// Mitsubishi GX Works2 project: js   PLC: Q02U
// js

PROGRAM MAIN
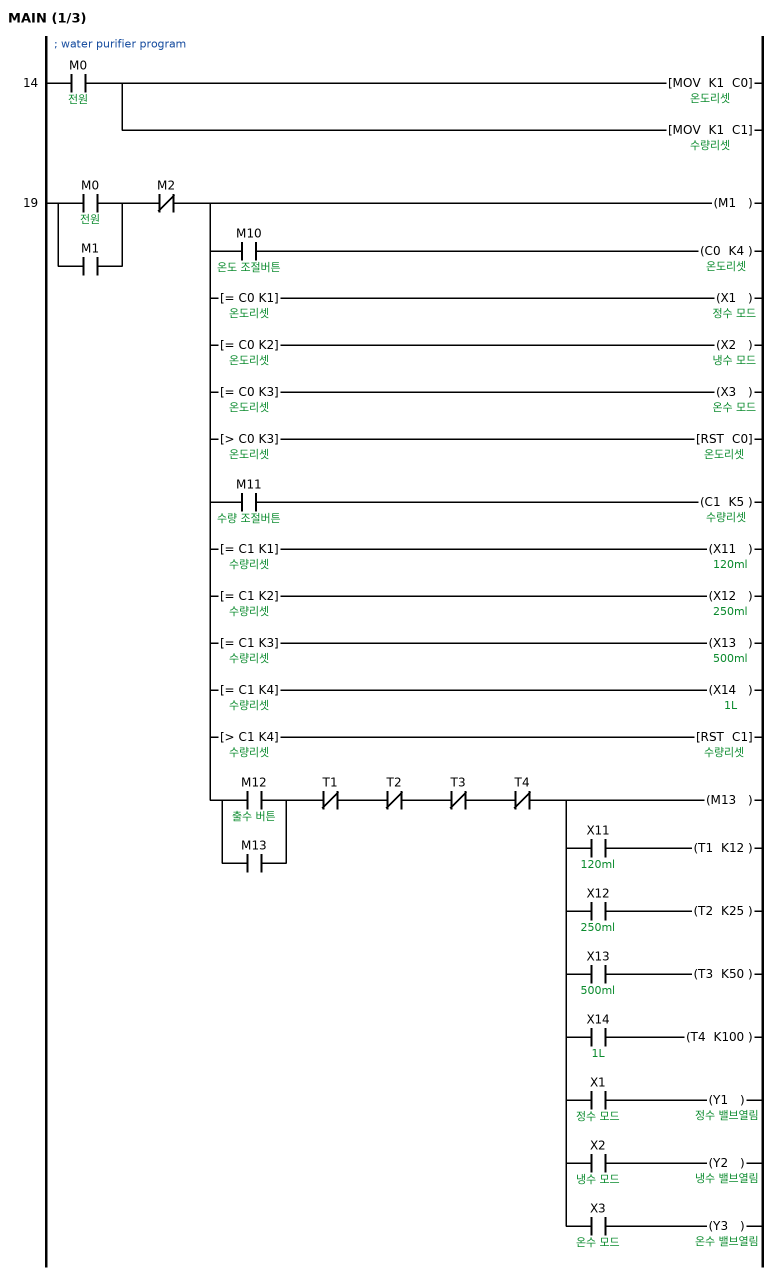
; water purifier program
14    LD      M0  ; 전원
      MOV     K1 C0  ; 온도리셋
      MOV     K1 C1  ; 수량리셋
19    LD      M0  ; 전원
      OR      M1
      ANI     M2
      OUT     M1
      MPS
      AND     M10  ; 온도 조절버튼
      OUT     C0 K4  ; 온도리셋
      MRD
      AND=    C0 K1  ; 온도리셋
      OUT     X1  ; 정수 모드
      MRD
      AND=    C0 K2  ; 온도리셋
      OUT     X2  ; 냉수 모드
      MRD
      AND=    C0 K3  ; 온도리셋
      OUT     X3  ; 온수 모드
      MRD
      AND>    C0 K3  ; 온도리셋
      RST     C0  ; 온도리셋
      MRD
      AND     M11  ; 수량 조절버튼
      OUT     C1 K5  ; 수량리셋
      MRD
      AND=    C1 K1  ; 수량리셋
      OUT     X11  ; 120ml
      MRD
      AND=    C1 K2  ; 수량리셋
      OUT     X12  ; 250ml
      MRD
      AND=    C1 K3  ; 수량리셋
      OUT     X13  ; 500ml
      MRD
      AND=    C1 K4  ; 수량리셋
      OUT     X14  ; 1L
      MRD
      AND>    C1 K4  ; 수량리셋
      RST     C1  ; 수량리셋
      MPP
      LD      M12  ; 출수 버튼
      OR      M13
      ANB
      ANI     T1
      ANI     T2
      ANI     T3
      ANI     T4
      OUT     M13
      MPS
      AND     X11  ; 120ml
      OUT     T1 K12
      MRD
      AND     X12  ; 250ml
      OUT     T2 K25
      MRD
      AND     X13  ; 500ml
      OUT     T3 K50
      MRD
      AND     X14  ; 1L
      OUT     T4 K100
      MRD
      AND     X1  ; 정수 모드
      OUT     Y1  ; 정수 밸브열림
      MRD
      AND     X2  ; 냉수 모드
      OUT     Y2  ; 냉수 밸브열림
      MPP
      AND     X3  ; 온수 모드
      OUT     Y3  ; 온수 밸브열림
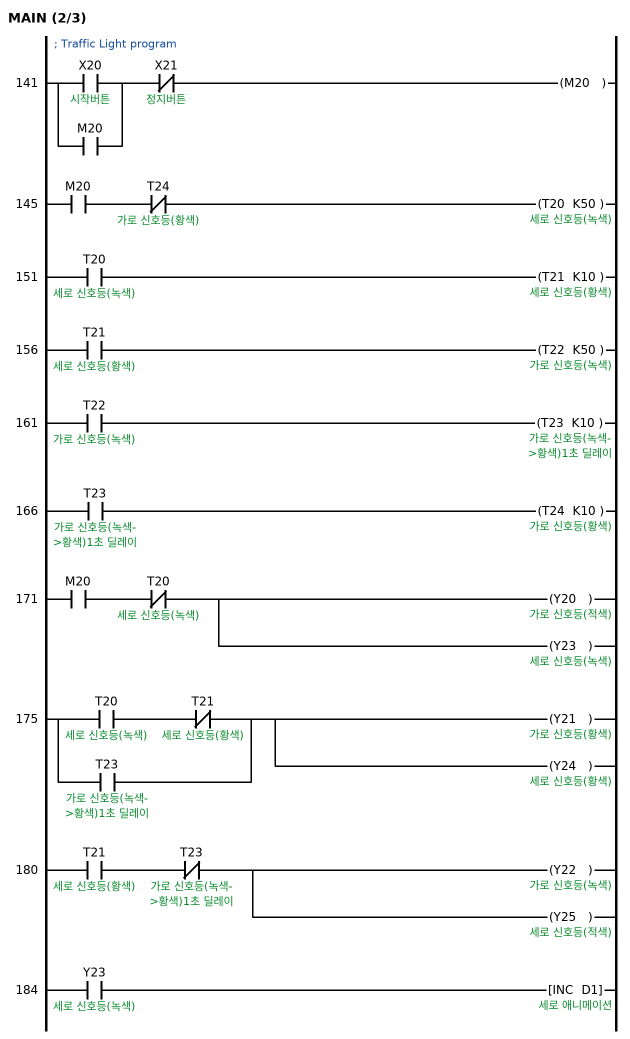
; Traffic Light program
141   LD      X20  ; 시작버튼
      OR      M20
      ANI     X21  ; 정지버튼
      OUT     M20
145   LD      M20
      ANI     T24  ; 가로 신호등(황색)
      OUT     T20 K50  ; 세로 신호등(녹색)
151   LD      T20  ; 세로 신호등(녹색)
      OUT     T21 K10  ; 세로 신호등(황색)
156   LD      T21  ; 세로 신호등(황색)
      OUT     T22 K50  ; 가로 신호등(녹색)
161   LD      T22  ; 가로 신호등(녹색)
      OUT     T23 K10  ; 가로 신호등(녹색->황색)1초 딜레이
166   LD      T23  ; 가로 신호등(녹색->황색)1초 딜레이
      OUT     T24 K10  ; 가로 신호등(황색)
171   LD      M20
      ANI     T20  ; 세로 신호등(녹색)
      OUT     Y20  ; 가로 신호등(적색)
      OUT     Y23  ; 세로 신호등(녹색)
175   LD      T20  ; 세로 신호등(녹색)
      ANI     T21  ; 세로 신호등(황색)
      OR      T23  ; 가로 신호등(녹색->황색)1초 딜레이
      OUT     Y21  ; 가로 신호등(황색)
      OUT     Y24  ; 세로 신호등(황색)
180   LD      T21  ; 세로 신호등(황색)
      ANI     T23  ; 가로 신호등(녹색->황색)1초 딜레이
      OUT     Y22  ; 가로 신호등(녹색)
      OUT     Y25  ; 세로 신호등(적색)
184   LD      Y23  ; 세로 신호등(녹색)
      INC     D1  ; 세로 애니메이션
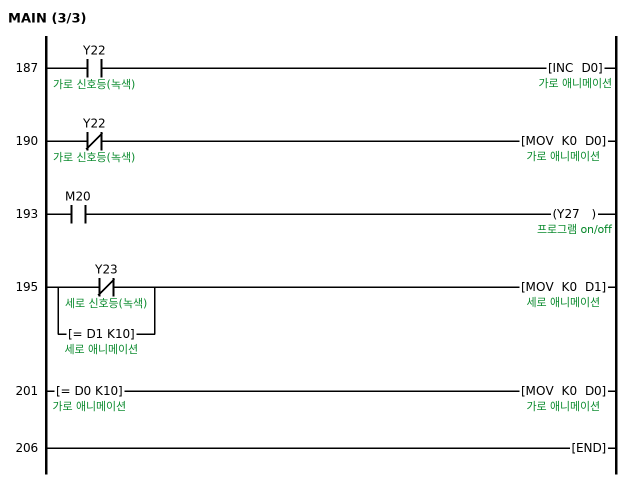
187   LD      Y22  ; 가로 신호등(녹색)
      INC     D0  ; 가로 애니메이션
190   LDI     Y22  ; 가로 신호등(녹색)
      MOV     K0 D0
193   LD      M20
      OUT     Y27  ; 프로그램 on/off
195   LDI     Y23  ; 세로 신호등(녹색)
      OR=     D1 K10  ; 세로 애니메이션
      MOV     K0 D1
201   LD=     D0 K10  ; 가로 애니메이션
      MOV     K0 D0
206   END
END_PROGRAM

// device comments not shown above
X22  ; 정지버튼
